// TIA Portal V18 export
// export: Created 2026-06-11T03:43:49.458617Z, ExportSetting WithDefaults, DisplayName Totally Integrated Automation Portal, DisplayVersion V18, DisplayName TIA Portal Openness, DisplayVersion V18, DisplayName TIA Portal Version Control Interface, DisplayVersion V18, DisplayName STEP 7 Professional, DisplayVersion V18, DisplayName STEP 7 Safety, DisplayVersion V18, DisplayName WinCC Professional, DisplayVersion V18
Screen "02_Van_Hanh"  800x600, Number=2
  ScreenLayer 
    GraphicView "Graphic view_1" at 0,0 size 800x600  Picture=Màn Vận Hành
    Button "Button_1" at 27,529 size 107x46  Mode=Text, TextOff="TỔNG QUAN", TextOn="Text"
      on Click: ActivateScreen(Screen name := 01_Tong_Quan, Object number := 0)
    Button "Button_3" at 281,529 size 107x46  Mode=Text, TextOff="PID MỨC", TextOn="Text"
      on Click: ActivateScreen(Screen name := 03_PID_Muc_Nuoc, Object number := 0)
    Button "Button_4" at 409,528 size 107x46  Mode=Text, TextOff="TREND", TextOn="Text"
      on Click: ActivateScreen(Screen name := 04_Trend, Object number := 0)
    Button "Button_5" at 537,528 size 107x46  Mode=Text, TextOff="CẢNH BÁO", TextOn="Text"
      on Click: ActivateScreen(Screen name := 05_Canh_Bao_IO, Object number := 0)
    TextField "Text field_1" at 249,3 size 285x31  Text="MÀN HÌNH 2 - VẬN HÀNH"
    Circle "Circle_3" at 677,3 size 39x39
      RangeAppearanceAnimation "RangeAppearanceAnimation"
        tag bSystemRun
        0..0: back #d9d9d9, fore #181c31
        1..1: back #00ff00, fore #181c31
    Circle "Circle_2" at 718,3 size 39x39
      RangeAppearanceAnimation "RangeAppearanceAnimation"
        tag Loi_He_Thong
        0..0: back #d9d9d9, fore #181c31
        1..1: back #ff0000, fore #181c31
    Circle "Circle_1" at 759,3 size 39x39
      RangeAppearanceAnimation "RangeAppearanceAnimation"
        tag bCheDoMoPhong
        0..0: back #d9d9d9, fore #181c31
        1..1: back #0000ff, fore #181c31
    TextField "Text field_2" at 679,42 size 34x22  Text="Run"
    TextField "Text field_3" at 717,42 size 43x22  Text="Fault"
    TextField "Text field_4" at 760,42 size 33x22  Text="Sim"
    TextField "Text field_5" at 57,69 size 131x22  Text="Bảng Điều Khiển"
    Button "Button_6" at 33,104 size 174x60  Mode=Text, TextOff="START", TextOn="Text"
      RangeAppearanceAnimation "RangeAppearanceAnimation"
        tag Nut_Start_HMI
        0..0: back #636571, fore #ffffff
        1..1: back #00ff00, fore #000000
      on Press: SetBit(Tag := Nut_Start_HMI)
      on Release: ResetBit(Tag := Nut_Start_HMI)
    Button "Button_7" at 33,178 size 174x60  Mode=Text, TextOff="STOP", TextOn="Text"
      RangeAppearanceAnimation "RangeAppearanceAnimation"
        tag Nut_Stop_HMI
        0..0: back #636571, fore #ffffff
        1..1: back #ff0000, fore #000000
      on Press: SetBit(Tag := Nut_Stop_HMI)
      on Release: ResetBit(Tag := Nut_Stop_HMI)
    Button "Button_8" at 33,252 size 174x60  Mode=Text, TextOff="RESET ALARM", TextOn="Text"
      RangeAppearanceAnimation "RangeAppearanceAnimation"
        tag Nut_Reset_HMI
        0..0: back #636571, fore #ffffff
        1..1: back #ffff00, fore #000000
      on Press: SetBit(Tag := Nut_Reset_HMI)
      on Release: ResetBit(Tag := Nut_Reset_HMI)
    Button "Button_9" at 33,327 size 174x60  Mode=Text, TextOff="SIMULATION", TextOn="Text"
      RangeAppearanceAnimation "RangeAppearanceAnimation"
        tag bCheDoMoPhong
        0..0: back #636571, fore #000000
        1..1: back #00ffff, fore #ffffff
      on Click: InvertBit(Tag := bCheDoMoPhong)
    Button "Button_10" at 33,402 size 174x60  Mode=Text, TextOff="E-STOP", TextOn="Text"
      RangeAppearanceAnimation "RangeAppearanceAnimation"
        tag Nut_EStop_HMI
        0..0: back #636571, fore #ffffff
        1..1: back #ff0000, fore #000000
      on Click: InvertBit(Tag := Nut_EStop_HMI)
    Rectangle "Rectangle_1" at 328,126 size 111x54
      RangeAppearanceAnimation "RangeAppearanceAnimation"
        tag Step0_IDLE
        0..0: back #d9d9d9, fore #181c31
        1..1: back #00ffff, fore #181c31
    Rectangle "Rectangle_2" at 328,206 size 111x53
      RangeAppearanceAnimation "RangeAppearanceAnimation"
        tag Step1_Thuc
        0..0: back #d9d9d9, fore #181c31
        1..1: back #ff6600, fore #181c31
    Rectangle "Rectangle_3" at 327,284 size 107x52
      RangeAppearanceAnimation "RangeAppearanceAnimation"
        tag Step2_Giu
        0..0: back #d9d9d9, fore #181c31
        1..1: back #339966, fore #181c31
    Rectangle "Rectangle_4" at 326,362 size 109x52
      RangeAppearanceAnimation "RangeAppearanceAnimation"
        tag Step3_KetThuc
        0..0: back #d9d9d9, fore #181c31
        1..1: back #333399, fore #181c31
    Rectangle "Rectangle_5" at 325,433 size 108x51
      RangeAppearanceAnimation "RangeAppearanceAnimation"
        tag StepErr_Loi
        0..0: back #d9d9d9, fore #181c31
        1..1: back #ff0000, fore #181c31, flashing
    TextField "Text field_6" at 333,145 size 97x18  Text="Chờ Khởi Động"
    TextField "Text field_7" at 332,225 size 102x18  Text="Gia Nhiệt Lò Hơi"
    TextField "Text field_8" at 331,302 size 97x18  Text="Chưng Cất PID"
    TextField "Text field_9" at 331,371 size 98x32  Text="Kết Thúc Và Hoàn Thành"
    TextField "Text field_10" at 336,450 size 86x18  Text="Lỗi Hệ Thống"
    Circle "Circle_4" at 590,83 size 38x38
      RangeAppearanceAnimation "RangeAppearanceAnimation"
        tag Den_Running_M
        0..0: back #d9d9d9, fore #181c31
        1..1: back #00ff00, fore #181c31
    Circle "Circle_5" at 591,132 size 38x38
      RangeAppearanceAnimation "RangeAppearanceAnimation"
        tag Van_Cap_Hoi_M
        0..0: back #d9d9d9, fore #181c31
        1..1: back #ff9900, fore #181c31
    Circle "Circle_6" at 591,181 size 38x38
      RangeAppearanceAnimation "RangeAppearanceAnimation"
        tag Bom_Lam_Mat_M
        0..0: back #d9d9d9, fore #181c31
        1..1: back #00ccff, fore #181c31
    Circle "Circle_7" at 591,230 size 38x38
      RangeAppearanceAnimation "RangeAppearanceAnimation"
        tag Bom_Hoan_Luu_M
        0..0: back #d9d9d9, fore #181c31
        1..1: back #d9d9d9, fore #0000ff
    Circle "Circle_8" at 591,279 size 38x38
      RangeAppearanceAnimation "RangeAppearanceAnimation"
        tag Coi_Alarm_M
        0..0: back #d9d9d9, fore #181c31
        1..1: back #ff0000, fore #181c31, flashing
    TextField "Text field_11" at 636,92 size 130x18  Text="Hệ thống đang chạy"
    TextField "Text field_12" at 651,141 size 99x18  Text="Van cấp hơi mở"
    TextField "Text field_13" at 641,190 size 120x18  Text="Bơm nước làm mát"
    TextField "Text field_14" at 654,239 size 91x18  Text="Bơm hoàn lưu"
    TextField "Text field_15" at 656,288 size 87x18  Text="Còi báo động"
    TextField "Text field_16" at 618,338 size 112x18  Text="Trạng thái chu kỳ"
    SymbolicIOField "Symbolic I/O field_1" at 585,358 size 184x37  CountVisibleItems=4, Mode=Output, OnValue=1, TextList=TL_VanHanh, TextOff="0", TextOn="1"
      ProcessValue := Main_State
    TextField "Text field_17" at 611,407 size 135x18  Text="Chuẩn Đoán An Toàn"
    SymbolicIOField "Symbolic I/O field_2" at 589,449 size 178x30  CountVisibleItems=3, Mode=Output, OnValue=1, TextList=TL_Chuan_Doan_AnToan, TextOff="0", TextOn="1"
      ProcessValue := HMI_Alarm_GFX
    Rectangle "Rectangle_8" at 149,526 size 114x52
    Button "Button_2" at 153,529 size 107x46  Mode=Text, TextOff="VẬN HÀNH", TextOn="Text"
      on Click: ActivateScreen(Screen name := , Object number := 0)
    Button "Button_11" at 732,552 size 65x30  Mode=Text, TextOff="EXIT", TextOn="Text"
      on Click: StopRuntime(Mode := 0)
    Button "Button_12" at 40,469 size 159x48  Mode=Text, TextOff="BOILER READY", TextOn="Text"
      RangeAppearanceAnimation "RangeAppearanceAnimation"
        tag Nut_Boiler_Ready_HMI
        0..0: back #636571, fore #ffffff
        1..1: back #00ccff, fore #000000
      on Click: InvertBit(Tag := Nut_Boiler_Ready_HMI)
